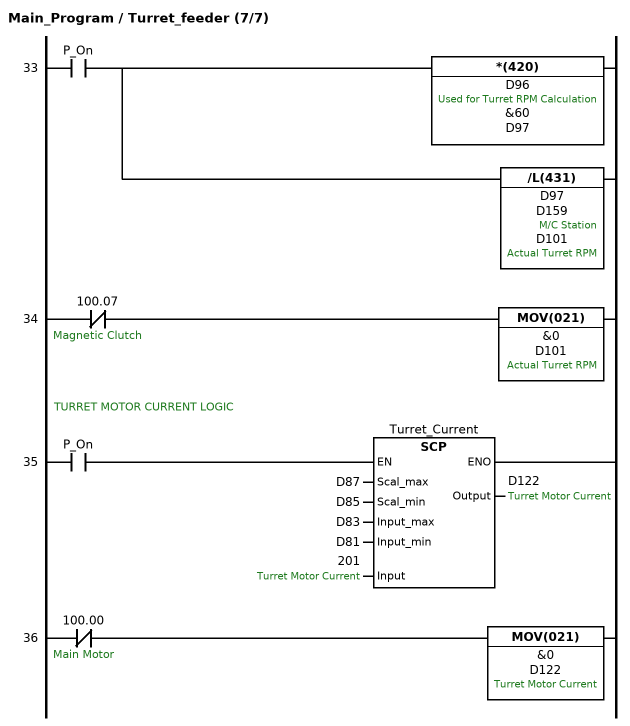
; [picture p24: Main_Program / Turret_feeder, rungs 33-36]
; rung 33
LD P_On
*(420) D96 &60 D97  ; Used for Turret RPM Calculation
/L(431) D97 D159 D101  ; M/C Station, Actual Turret RPM
; rung 34
LDNOT 100.07  ; Magnetic Clutch
MOV(021) &0 D101  ; Actual Turret RPM
; rung 35: TURRET MOTOR CURRENT LOGIC
LD P_On
CALL Turret_Current : SCP (Scal_max := D87, Scal_min := D85, Input_max := D83, Input_min := D81, Input := 201, Output => D122)  ; Turret Motor Current
; rung 36
LDNOT 100.00  ; Main Motor
MOV(021) &0 D122  ; Turret Motor Current

### Section Hyd_System
; Main Hyd. System Pressure

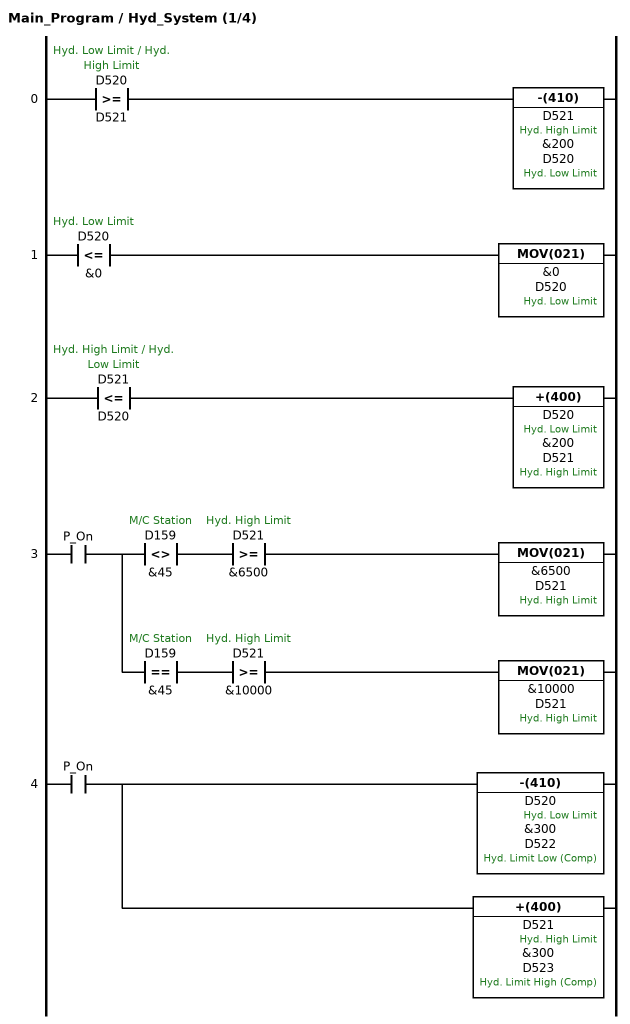
; rung 0
LD>=(325) D520 D521  ; Hyd. Low Limit, Hyd. High Limit
-(410) D521 &200 D520  ; Hyd. High Limit, Hyd. Low Limit
; rung 1
LD<=S(317) D520 &0  ; Hyd. Low Limit
MOV(021) &0 D520  ; Hyd. Low Limit
; rung 2
LD<=(315) D521 D520  ; Hyd. High Limit, Hyd. Low Limit
+(400) D520 &200 D521  ; Hyd. Low Limit, Hyd. High Limit
; rung 3
LD P_On
OUT TR0
AND<>(305) D159 &45  ; M/C Station
AND>=(325) D521 &6500  ; Hyd. High Limit
MOV(021) &6500 D521  ; Hyd. High Limit
LD TR0
AND=(300) D159 &45  ; M/C Station
AND>=(325) D521 &10000  ; Hyd. High Limit
MOV(021) &10000 D521  ; Hyd. High Limit
; rung 4
LD P_On
-(410) D520 &300 D522  ; Hyd. Low Limit, Hyd. Limit Low (Comp)
+(400) D521 &300 D523  ; Hyd. High Limit, Hyd. Limit High (Comp)

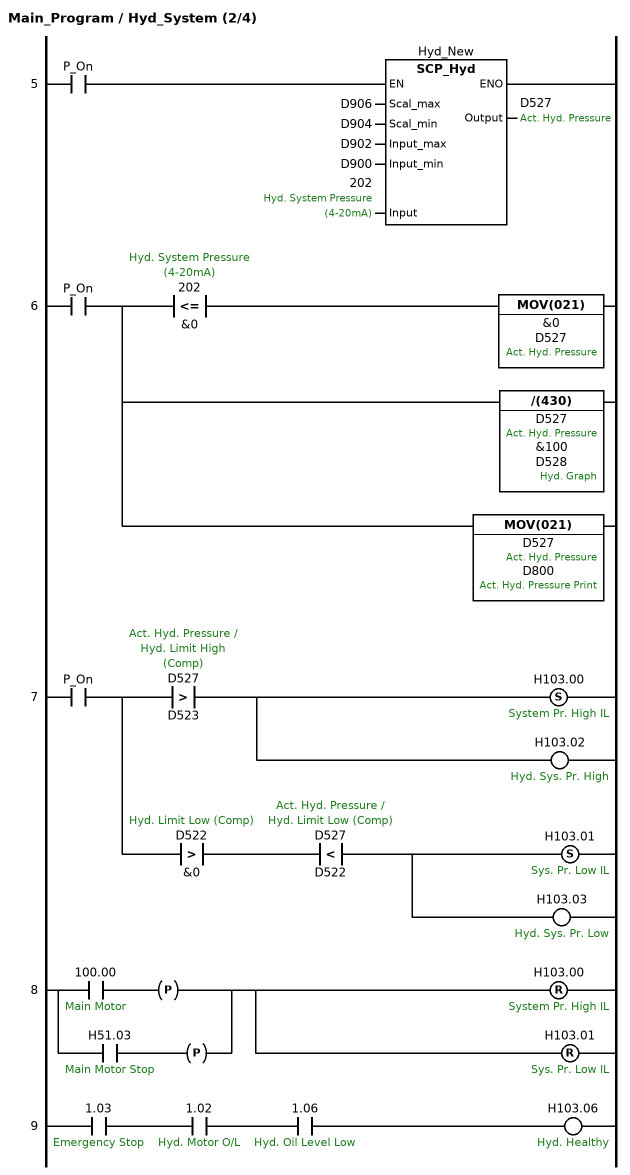
; rung 5
LD P_On
CALL Hyd_New : SCP_Hyd (Scal_max := D906, Scal_min := D904, Input_max := D902, Input_min := D900, Input := 202, Output => D527)  ; Hyd. System Pressure (4-20mA), Act. Hyd. Pressure
; rung 6
LD P_On
OUT TR0
AND<=S(317) 202 &0  ; Hyd. System Pressure (4-20mA)
MOV(021) &0 D527  ; Act. Hyd. Pressure
LD TR0
/(430) D527 &100 D528  ; Act. Hyd. Pressure, Hyd. Graph
MOV(021) D527 D800  ; Act. Hyd. Pressure, Act. Hyd. Pressure Print
; rung 7
LD P_On
OUT TR0
AND>(320) D527 D523  ; Act. Hyd. Pressure, Hyd. Limit High (Comp)
SET H103.00  ; System Pr. High IL
OUT H103.02  ; Hyd. Sys. Pr. High
LD TR0
AND>S(322) D522 &0  ; Hyd. Limit Low (Comp)
AND<(310) D527 D522  ; Act. Hyd. Pressure, Hyd. Limit Low (Comp)
SET H103.01  ; Sys. Pr. Low IL
OUT H103.03  ; Hyd. Sys. Pr. Low
; rung 8
LD 100.00  ; Main Motor
UP(521)
LD H51.03  ; Main Motor Stop
UP(521)
ORLD
RSET H103.00  ; System Pr. High IL
RSET H103.01  ; Sys. Pr. Low IL
; rung 9
LD 1.03  ; Emergency Stop
AND 1.02  ; Hyd. Motor O/L
AND 1.06  ; Hyd. Oil Level Low
OUT H103.06  ; Hyd. Healthy

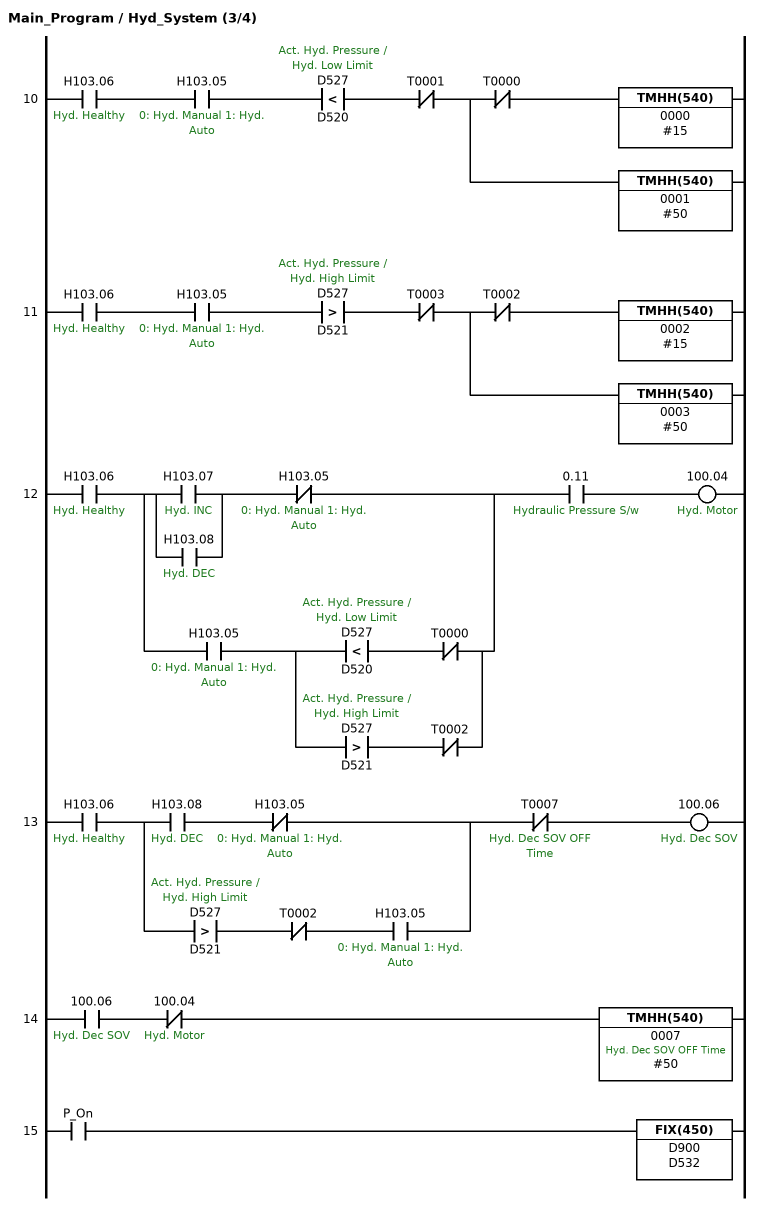
; rung 10
LD H103.06  ; Hyd. Healthy
AND H103.05  ; 0: Hyd. Manual 1: Hyd. Auto
AND<(310) D527 D520  ; Act. Hyd. Pressure, Hyd. Low Limit
ANDNOT T0001
OUT TR0
ANDNOT T0000
TMHH(540) 0000 #15
LD TR0
TMHH(540) 0001 #50
; rung 11
LD H103.06  ; Hyd. Healthy
AND H103.05  ; 0: Hyd. Manual 1: Hyd. Auto
AND>(320) D527 D521  ; Act. Hyd. Pressure, Hyd. High Limit
ANDNOT T0003
OUT TR0
ANDNOT T0002
TMHH(540) 0002 #15
LD TR0
TMHH(540) 0003 #50
; rung 12
LD H103.06  ; Hyd. Healthy
LD H103.07  ; Hyd. INC
OR H103.08  ; Hyd. DEC
ANDNOT H103.05  ; 0: Hyd. Manual 1: Hyd. Auto
LD H103.05  ; 0: Hyd. Manual 1: Hyd. Auto
LD<(310) D527 D520  ; Act. Hyd. Pressure, Hyd. Low Limit
ANDNOT T0000
LD>(320) D527 D521  ; Act. Hyd. Pressure, Hyd. High Limit
ANDNOT T0002
ORLD
ANDLD
ORLD
ANDLD
AND 0.11  ; Hydraulic Pressure S/w
OUT 100.04  ; Hyd. Motor
; rung 13
LD H103.06  ; Hyd. Healthy
LD H103.08  ; Hyd. DEC
ANDNOT H103.05  ; 0: Hyd. Manual 1: Hyd. Auto
LD>(320) D527 D521  ; Act. Hyd. Pressure, Hyd. High Limit
ANDNOT T0002
AND H103.05  ; 0: Hyd. Manual 1: Hyd. Auto
ORLD
ANDLD
ANDNOT T0007  ; Hyd. Dec SOV OFF Time
OUT 100.06  ; Hyd. Dec SOV
; rung 14
LD 100.06  ; Hyd. Dec SOV
ANDNOT 100.04  ; Hyd. Motor
TMHH(540) 0007 #50  ; Hyd. Dec SOV OFF Time
; rung 15
LD P_On
FIX(450) D900 D532

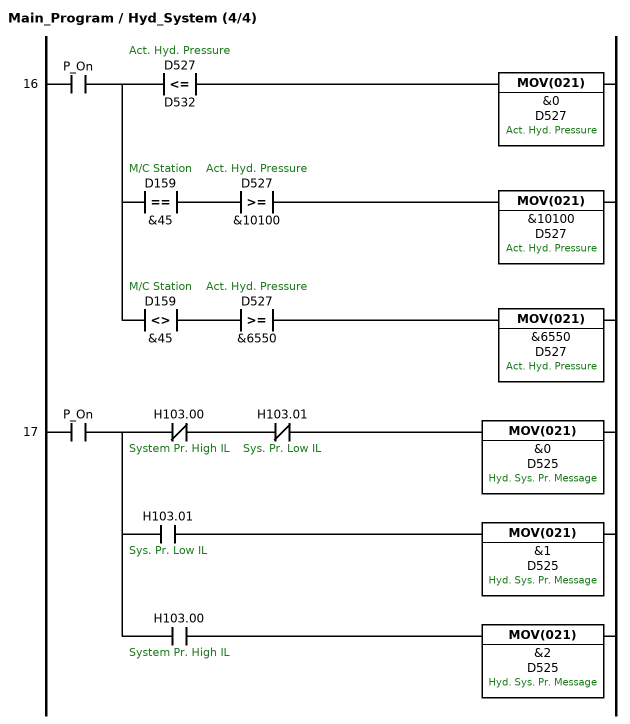
; rung 16
LD P_On
OUT TR0
AND<=(315) D527 D532  ; Act. Hyd. Pressure
MOV(021) &0 D527  ; Act. Hyd. Pressure
LD TR0
AND=(300) D159 &45  ; M/C Station
AND>=(325) D527 &10100  ; Act. Hyd. Pressure
MOV(021) &10100 D527  ; Act. Hyd. Pressure
LD TR0
AND<>(305) D159 &45  ; M/C Station
AND>=(325) D527 &6550  ; Act. Hyd. Pressure
MOV(021) &6550 D527  ; Act. Hyd. Pressure
; rung 17
LD P_On
OUT TR0
ANDNOT H103.00  ; System Pr. High IL
ANDNOT H103.01  ; Sys. Pr. Low IL
MOV(021) &0 D525  ; Hyd. Sys. Pr. Message
LD TR0
AND H103.01  ; Sys. Pr. Low IL
MOV(021) &1 D525  ; Hyd. Sys. Pr. Message
LD TR0
AND H103.00  ; System Pr. High IL
MOV(021) &2 D525  ; Hyd. Sys. Pr. Message

### Section Lubrication
; Lubrication Control & Hour Meter

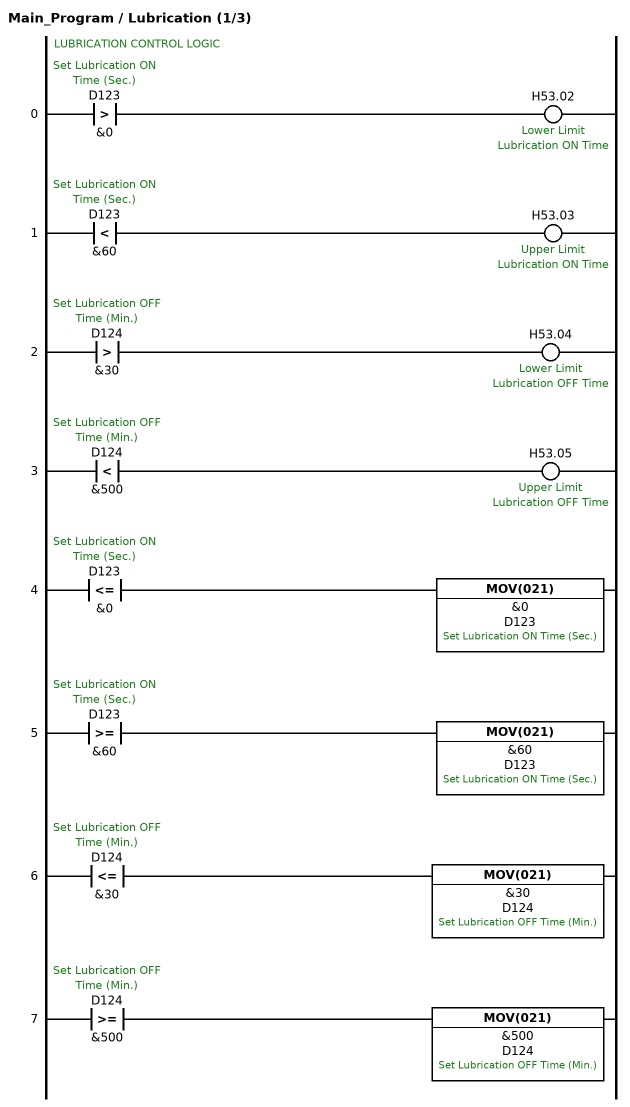
; rung 0: LUBRICATION CONTROL LOGIC
LD>(320) D123 &0  ; Set Lubrication ON Time (Sec.)
OUT H53.02  ; Lower Limit Lubrication ON Time
; rung 1
LD<(310) D123 &60  ; Set Lubrication ON Time (Sec.)
OUT H53.03  ; Upper Limit Lubrication ON Time
; rung 2
LD>(320) D124 &30  ; Set Lubrication OFF Time (Min.)
OUT H53.04  ; Lower Limit Lubrication OFF Time
; rung 3
LD<(310) D124 &500  ; Set Lubrication OFF Time (Min.)
OUT H53.05  ; Upper Limit Lubrication OFF Time
; rung 4
LD<=(315) D123 &0  ; Set Lubrication ON Time (Sec.)
MOV(021) &0 D123  ; Set Lubrication ON Time (Sec.)
; rung 5
LD>=(325) D123 &60  ; Set Lubrication ON Time (Sec.)
MOV(021) &60 D123  ; Set Lubrication ON Time (Sec.)
; rung 6
LD<=(315) D124 &30  ; Set Lubrication OFF Time (Min.)
MOV(021) &30 D124  ; Set Lubrication OFF Time (Min.)
; rung 7
LD>=(325) D124 &500  ; Set Lubrication OFF Time (Min.)
MOV(021) &500 D124  ; Set Lubrication OFF Time (Min.)

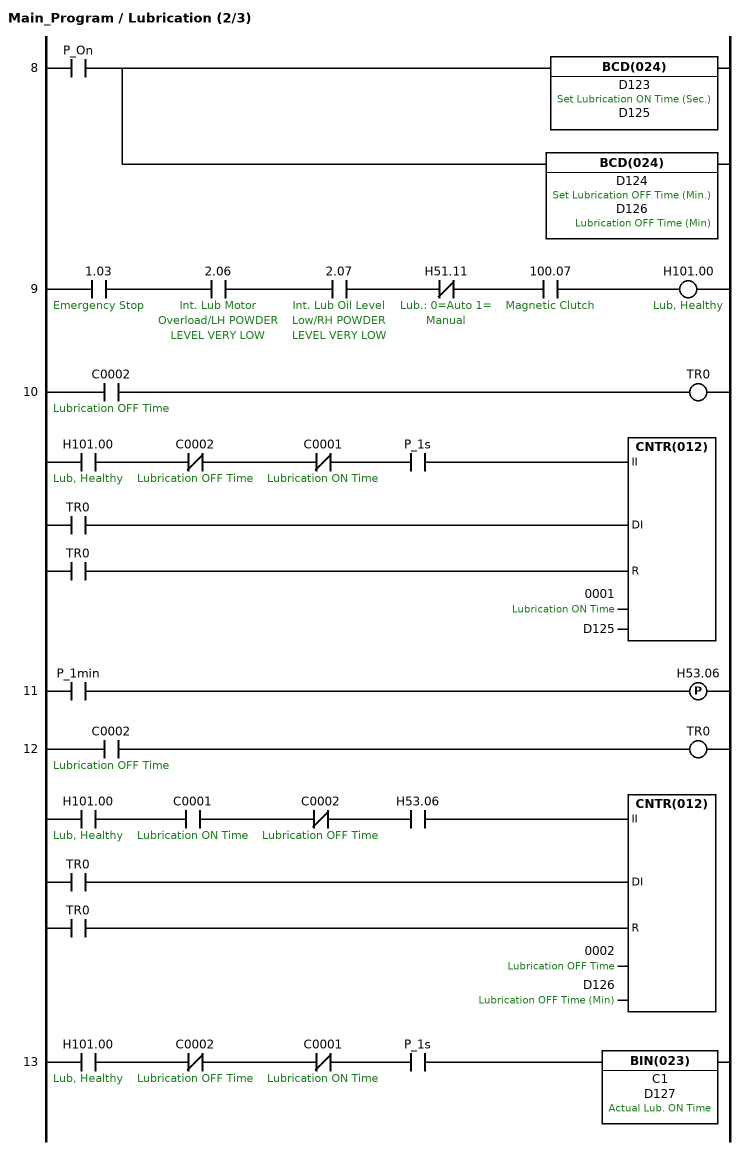
; rung 8
LD P_On
BCD(024) D123 D125  ; Set Lubrication ON Time (Sec.)
BCD(024) D124 D126  ; Set Lubrication OFF Time (Min.), Lubrication OFF Time (Min)
; rung 9
LD 1.03  ; Emergency Stop
AND 2.06  ; Int. Lub Motor Overload/LH POWDER LEVEL VERY LOW
AND 2.07  ; Int. Lub Oil Level Low/RH POWDER LEVEL VERY LOW
ANDNOT H51.11  ; Lub.: 0=Auto 1= Manual
AND 100.07  ; Magnetic Clutch
OUT H101.00  ; Lub, Healthy
; rung 10
LD H101.00  ; Lub, Healthy
ANDNOT C0002  ; Lubrication OFF Time
ANDNOT C0001  ; Lubrication ON Time
AND P_1s
LD C0002  ; Lubrication OFF Time
OUT TR0
LD TR0
CNTR(012) 0001 D125  ; Lubrication ON Time
; rung 11
LD P_1min
DIFU(013) H53.06
; rung 12
LD H101.00  ; Lub, Healthy
AND C0001  ; Lubrication ON Time
ANDNOT C0002  ; Lubrication OFF Time
AND H53.06
LD C0002  ; Lubrication OFF Time
OUT TR0
LD TR0
CNTR(012) 0002 D126  ; Lubrication OFF Time (Min), Lubrication OFF Time
; rung 13
LD H101.00  ; Lub, Healthy
ANDNOT C0002  ; Lubrication OFF Time
ANDNOT C0001  ; Lubrication ON Time
AND P_1s
BIN(023) C1 D127  ; Actual Lub. ON Time

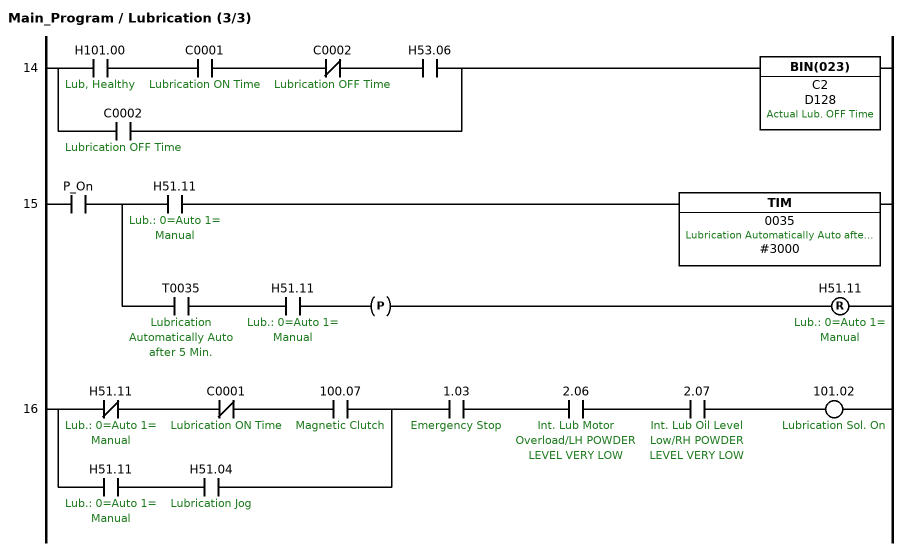
; rung 14
LD H101.00  ; Lub, Healthy
AND C0001  ; Lubrication ON Time
ANDNOT C0002  ; Lubrication OFF Time
AND H53.06
OR C0002  ; Lubrication OFF Time
BIN(023) C2 D128  ; Actual Lub. OFF Time
; rung 15
LD P_On
OUT TR0
AND H51.11  ; Lub.: 0=Auto 1= Manual
TIM 0035 #3000  ; Lubrication Automatically Auto after 5 Min.
LD TR0
AND T0035  ; Lubrication Automatically Auto after 5 Min.
AND H51.11  ; Lub.: 0=Auto 1= Manual
UP(521)
RSET H51.11  ; Lub.: 0=Auto 1= Manual
; rung 16
LDNOT H51.11  ; Lub.: 0=Auto 1= Manual
ANDNOT C0001  ; Lubrication ON Time
AND 100.07  ; Magnetic Clutch
LD H51.11  ; Lub.: 0=Auto 1= Manual
AND H51.04  ; Lubrication Jog
ORLD
AND 1.03  ; Emergency Stop
AND 2.06  ; Int. Lub Motor Overload/LH POWDER LEVEL VERY LOW
AND 2.07  ; Int. Lub Oil Level Low/RH POWDER LEVEL VERY LOW
OUT 101.02  ; Lubrication Sol. On

### Section LPSL
; Lower Punch Spray Control

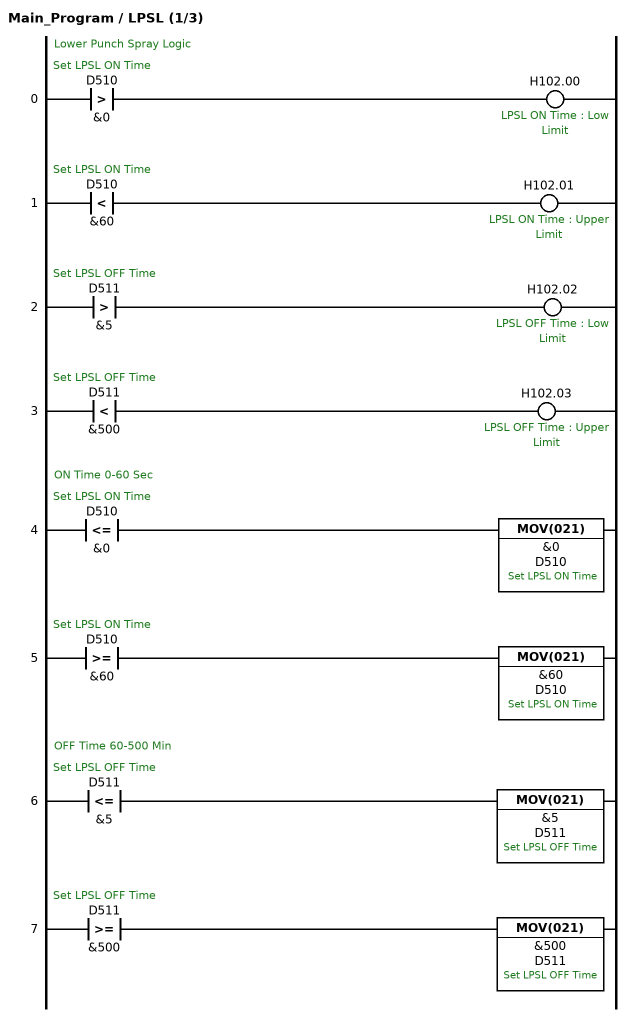
; rung 0: Lower Punch Spray Logic
LD>(320) D510 &0  ; Set LPSL ON Time
OUT H102.00  ; LPSL ON Time : Low Limit
; rung 1
LD<(310) D510 &60  ; Set LPSL ON Time
OUT H102.01  ; LPSL ON Time : Upper Limit
; rung 2
LD>(320) D511 &5  ; Set LPSL OFF Time
OUT H102.02  ; LPSL OFF Time : Low Limit
; rung 3
LD<(310) D511 &500  ; Set LPSL OFF Time
OUT H102.03  ; LPSL OFF Time : Upper Limit
; rung 4: ON Time 0-60 Sec
LD<=(315) D510 &0  ; Set LPSL ON Time
MOV(021) &0 D510  ; Set LPSL ON Time
; rung 5
LD>=(325) D510 &60  ; Set LPSL ON Time
MOV(021) &60 D510  ; Set LPSL ON Time
; rung 6: OFF Time 60-500 Min
LD<=(315) D511 &5  ; Set LPSL OFF Time
MOV(021) &5 D511  ; Set LPSL OFF Time
; rung 7
LD>=(325) D511 &500  ; Set LPSL OFF Time
MOV(021) &500 D511  ; Set LPSL OFF Time

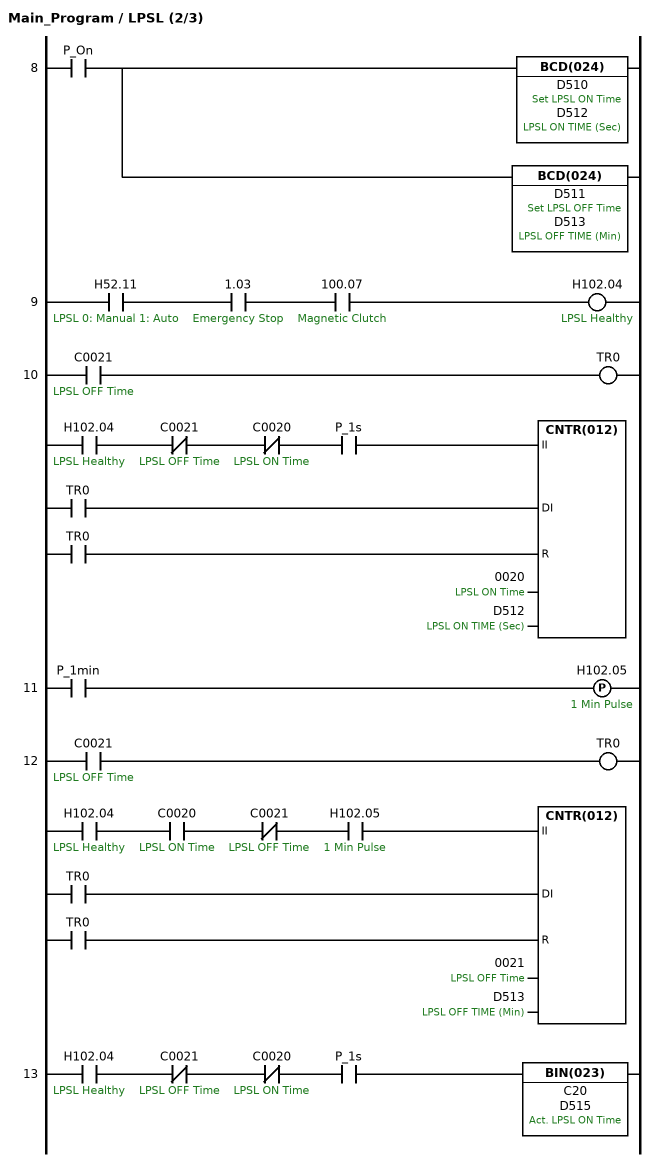
; rung 8
LD P_On
BCD(024) D510 D512  ; Set LPSL ON Time, LPSL ON TIME (Sec)
BCD(024) D511 D513  ; Set LPSL OFF Time, LPSL OFF TIME (Min)
; rung 9
LD H52.11  ; LPSL 0: Manual 1: Auto
AND 1.03  ; Emergency Stop
AND 100.07  ; Magnetic Clutch
OUT H102.04  ; LPSL Healthy
; rung 10
LD H102.04  ; LPSL Healthy
ANDNOT C0021  ; LPSL OFF Time
ANDNOT C0020  ; LPSL ON Time
AND P_1s
LD C0021  ; LPSL OFF Time
OUT TR0
LD TR0
CNTR(012) 0020 D512  ; LPSL ON TIME (Sec), LPSL ON Time
; rung 11
LD P_1min
DIFU(013) H102.05  ; 1 Min Pulse
; rung 12
LD H102.04  ; LPSL Healthy
AND C0020  ; LPSL ON Time
ANDNOT C0021  ; LPSL OFF Time
AND H102.05  ; 1 Min Pulse
LD C0021  ; LPSL OFF Time
OUT TR0
LD TR0
CNTR(012) 0021 D513  ; LPSL OFF TIME (Min), LPSL OFF Time
; rung 13
LD H102.04  ; LPSL Healthy
ANDNOT C0021  ; LPSL OFF Time
ANDNOT C0020  ; LPSL ON Time
AND P_1s
BIN(023) C20 D515  ; Act. LPSL ON Time

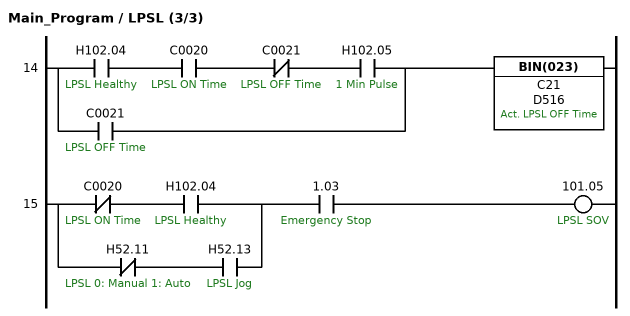
; rung 14
LD H102.04  ; LPSL Healthy
AND C0020  ; LPSL ON Time
ANDNOT C0021  ; LPSL OFF Time
AND H102.05  ; 1 Min Pulse
OR C0021  ; LPSL OFF Time
BIN(023) C21 D516  ; Act. LPSL OFF Time
; rung 15
LDNOT C0020  ; LPSL ON Time
AND H102.04  ; LPSL Healthy
LDNOT H52.11  ; LPSL 0: Manual 1: Auto
AND H52.13  ; LPSL Jog
ORLD
AND 1.03  ; Emergency Stop
OUT 101.05  ; LPSL SOV

### Section Agitator

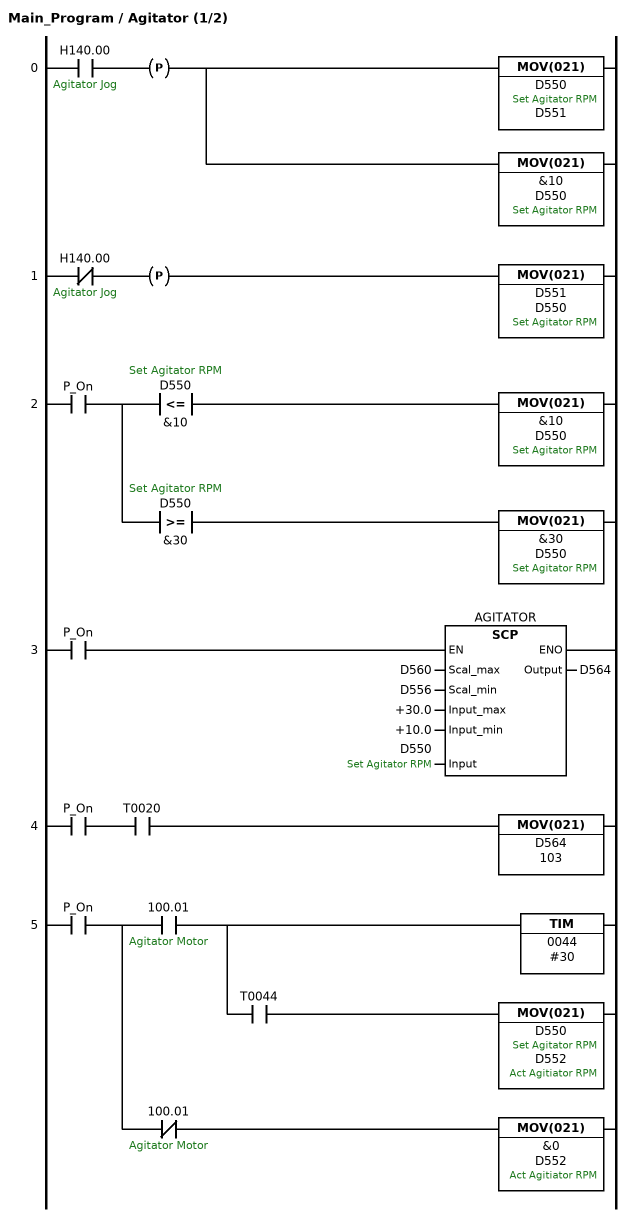
; rung 0
LD H140.00  ; Agitator Jog
UP(521)
MOV(021) D550 D551  ; Set Agitator RPM
MOV(021) &10 D550  ; Set Agitator RPM
; rung 1
LDNOT H140.00  ; Agitator Jog
UP(521)
MOV(021) D551 D550  ; Set Agitator RPM
; rung 2
LD P_On
OUT TR0
AND<=(315) D550 &10  ; Set Agitator RPM
MOV(021) &10 D550  ; Set Agitator RPM
LD TR0
AND>=(325) D550 &30  ; Set Agitator RPM
MOV(021) &30 D550  ; Set Agitator RPM
; rung 3
LD P_On
CALL AGITATOR : SCP (Scal_max := D560, Scal_min := D556, Input_max := +30.0, Input_min := +10.0, Input := D550, Output => D564)  ; Set Agitator RPM
; rung 4
LD P_On
AND T0020
MOV(021) D564 103
; rung 5
LD P_On
OUT TR0
AND 100.01  ; Agitator Motor
TIM 0044 #30
AND T0044
MOV(021) D550 D552  ; Set Agitator RPM, Act Agitiator RPM
LD TR0
ANDNOT 100.01  ; Agitator Motor
MOV(021) &0 D552  ; Act Agitiator RPM

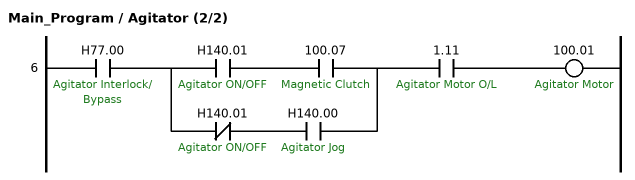
; rung 6
LD H77.00  ; Agitator Interlock/Bypass
LD H140.01  ; Agitator ON/OFF
AND 100.07  ; Magnetic Clutch
LDNOT H140.01  ; Agitator ON/OFF
AND H140.00  ; Agitator Jog
ORLD
ANDLD
AND 1.11  ; Agitator Motor O/L
OUT 100.01  ; Agitator Motor

### Section Recipe

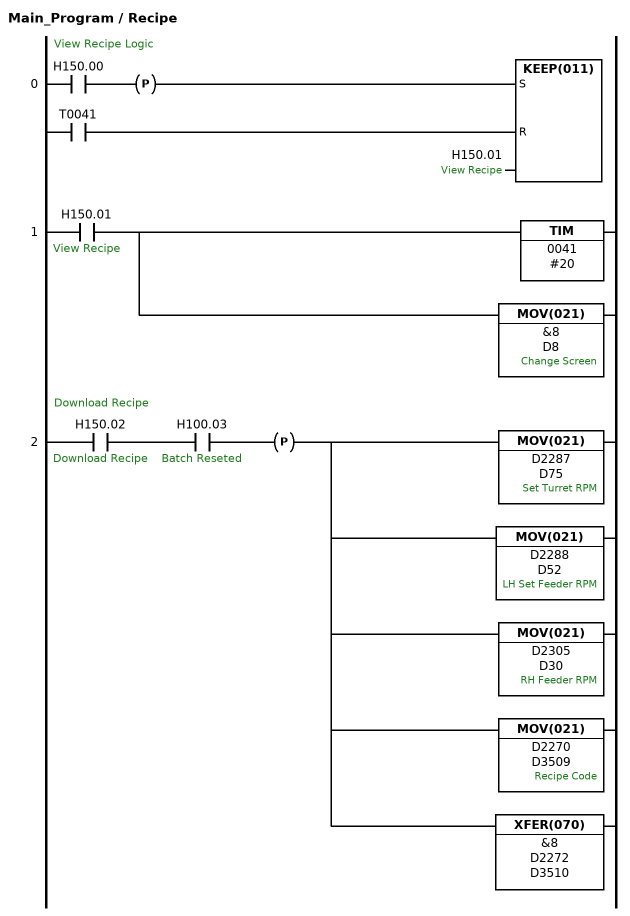
; rung 0: View Recipe Logic
LD H150.00
UP(521)
LD T0041
KEEP(011) H150.01  ; View Recipe
; rung 1
LD H150.01  ; View Recipe
TIM 0041 #20
MOV(021) &8 D8  ; Change Screen
; rung 2: Download Recipe
LD H150.02  ; Download Recipe
AND H100.03  ; Batch Reseted
UP(521)
MOV(021) D2287 D75  ; Set Turret RPM
MOV(021) D2288 D52  ; LH Set Feeder RPM
MOV(021) D2305 D30  ; RH Feeder RPM
MOV(021) D2270 D3509  ; Recipe Code
XFER(070) &8 D2272 D3510

### Section Interlock

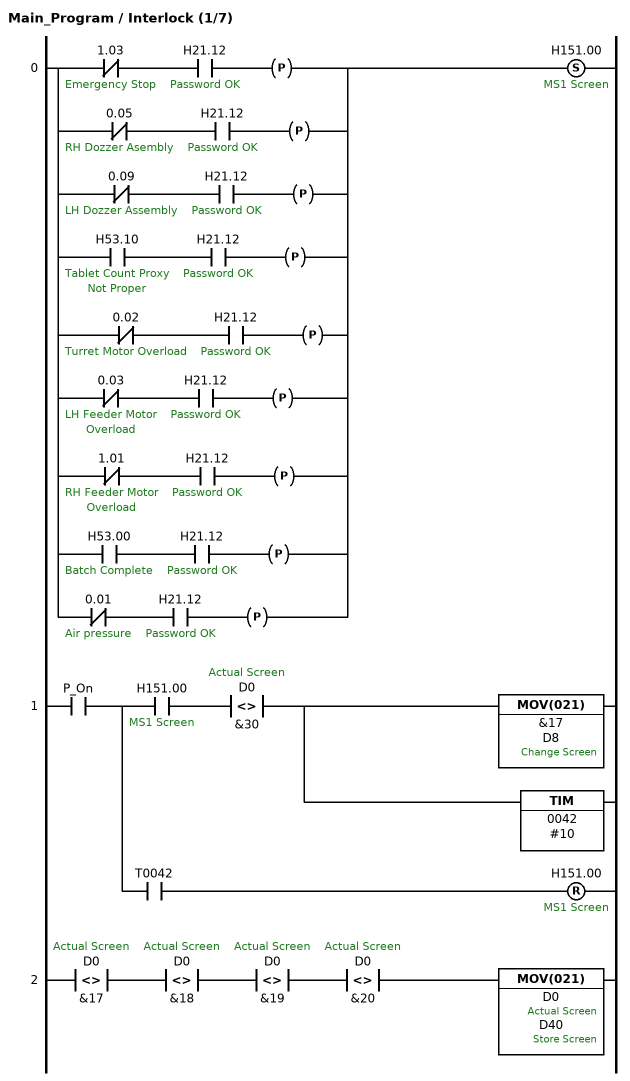
; rung 0
LDNOT 1.03  ; Emergency Stop
AND H21.12  ; Password OK
UP(521)
LDNOT 0.05  ; RH Dozzer Asembly
AND H21.12  ; Password OK
UP(521)
ORLD
LDNOT 0.09  ; LH Dozzer Assembly
AND H21.12  ; Password OK
UP(521)
ORLD
LD H53.10  ; Tablet Count Proxy Not Proper
AND H21.12  ; Password OK
UP(521)
ORLD
LDNOT 0.02  ; Turret Motor Overload
AND H21.12  ; Password OK
UP(521)
ORLD
LDNOT 0.03  ; LH Feeder Motor Overload
AND H21.12  ; Password OK
UP(521)
ORLD
LDNOT 1.01  ; RH Feeder Motor Overload
AND H21.12  ; Password OK
UP(521)
ORLD
LD H53.00  ; Batch Complete
AND H21.12  ; Password OK
UP(521)
ORLD
LDNOT 0.01  ; Air pressure
AND H21.12  ; Password OK
UP(521)
ORLD
SET H151.00  ; MS1 Screen
; rung 1
LD P_On
OUT TR0
AND H151.00  ; MS1 Screen
AND<>(305) D0 &30  ; Actual Screen
MOV(021) &17 D8  ; Change Screen
TIM 0042 #10
LD TR0
AND T0042
RSET H151.00  ; MS1 Screen
; rung 2
LD<>(305) D0 &17  ; Actual Screen
AND<>(305) D0 &18  ; Actual Screen
AND<>(305) D0 &19  ; Actual Screen
AND<>(305) D0 &20  ; Actual Screen
MOV(021) D0 D40  ; Actual Screen, Store Screen

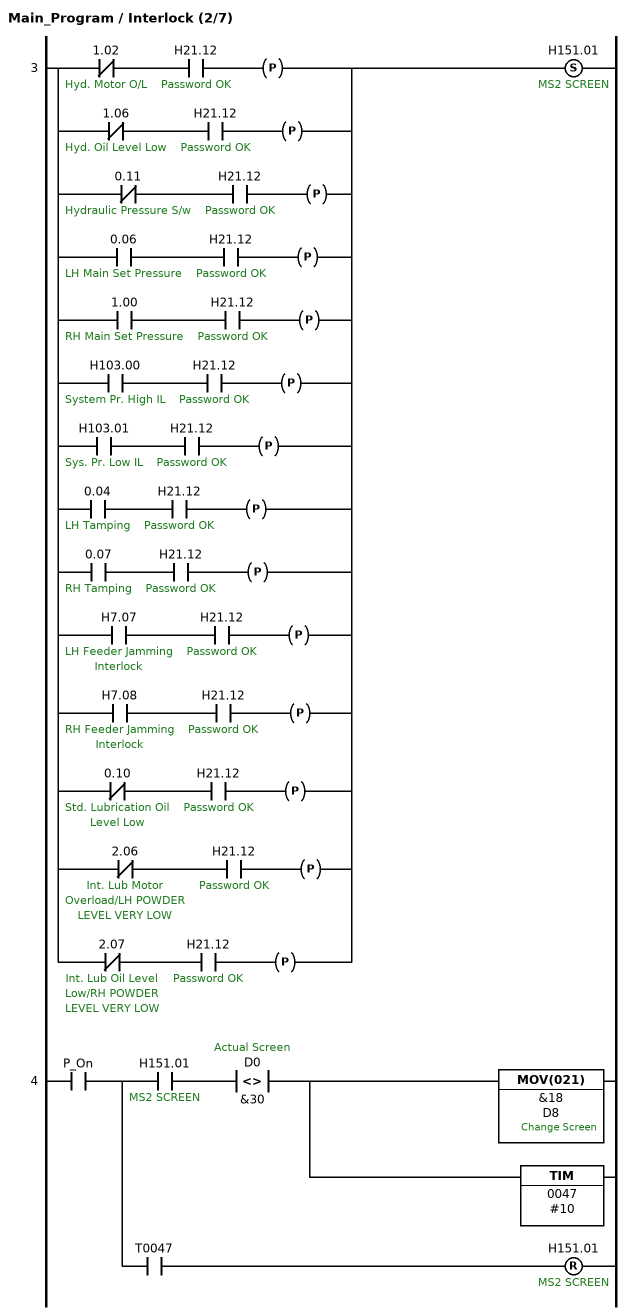
; rung 3
LDNOT 1.02  ; Hyd. Motor O/L
AND H21.12  ; Password OK
UP(521)
LDNOT 1.06  ; Hyd. Oil Level Low
AND H21.12  ; Password OK
UP(521)
ORLD
LDNOT 0.11  ; Hydraulic Pressure S/w
AND H21.12  ; Password OK
UP(521)
ORLD
LD 0.06  ; LH Main Set Pressure
AND H21.12  ; Password OK
UP(521)
ORLD
LD 1.00  ; RH Main Set Pressure
AND H21.12  ; Password OK
UP(521)
ORLD
LD H103.00  ; System Pr. High IL
AND H21.12  ; Password OK
UP(521)
ORLD
LD H103.01  ; Sys. Pr. Low IL
AND H21.12  ; Password OK
UP(521)
ORLD
LD 0.04  ; LH Tamping
AND H21.12  ; Password OK
UP(521)
ORLD
LD 0.07  ; RH Tamping
AND H21.12  ; Password OK
UP(521)
ORLD
LD H7.07  ; LH Feeder Jamming Interlock
AND H21.12  ; Password OK
UP(521)
ORLD
LD H7.08  ; RH Feeder Jamming Interlock
AND H21.12  ; Password OK
UP(521)
ORLD
LDNOT 0.10  ; Std. Lubrication Oil Level Low
AND H21.12  ; Password OK
UP(521)
ORLD
LDNOT 2.06  ; Int. Lub Motor Overload/LH POWDER LEVEL VERY LOW
AND H21.12  ; Password OK
UP(521)
ORLD
LDNOT 2.07  ; Int. Lub Oil Level Low/RH POWDER LEVEL VERY LOW
AND H21.12  ; Password OK
UP(521)
ORLD
SET H151.01  ; MS2 SCREEN
; rung 4
LD P_On
OUT TR0
AND H151.01  ; MS2 SCREEN
AND<>(305) D0 &30  ; Actual Screen
MOV(021) &18 D8  ; Change Screen
TIM 0047 #10
LD TR0
AND T0047
RSET H151.01  ; MS2 SCREEN

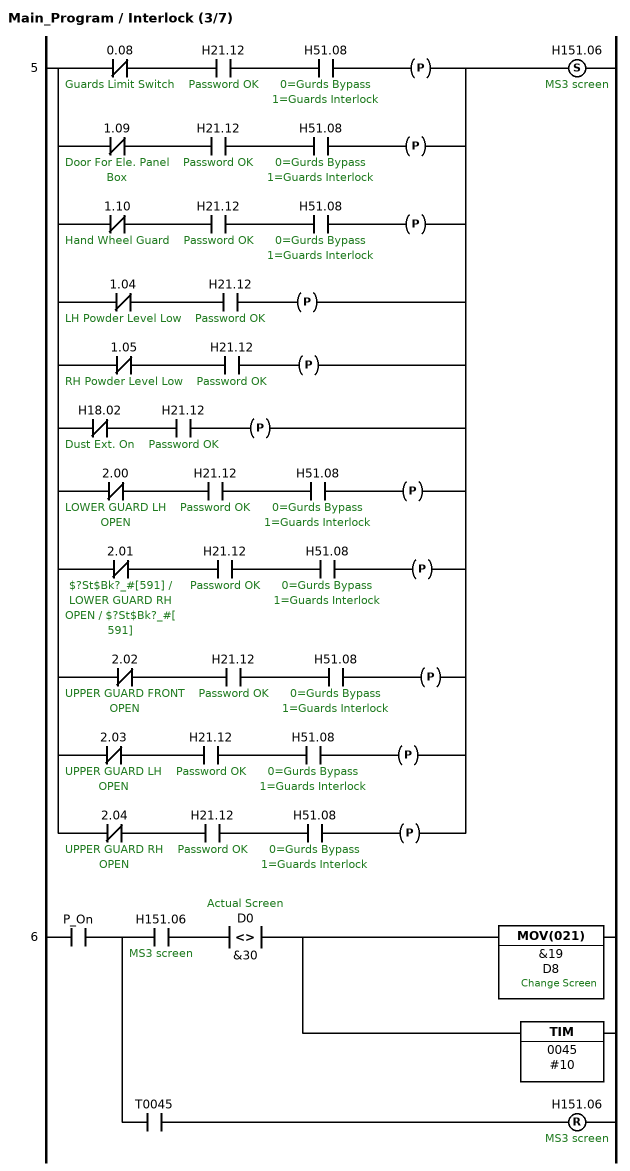
; rung 5
LDNOT 0.08  ; Guards Limit Switch
AND H21.12  ; Password OK
AND H51.08  ; 0=Gurds Bypass 1=Guards Interlock
UP(521)
LDNOT 1.09  ; Door For Ele. Panel Box
AND H21.12  ; Password OK
AND H51.08  ; 0=Gurds Bypass 1=Guards Interlock
UP(521)
ORLD
LDNOT 1.10  ; Hand Wheel Guard
AND H21.12  ; Password OK
AND H51.08  ; 0=Gurds Bypass 1=Guards Interlock
UP(521)
ORLD
LDNOT 1.04  ; LH Powder Level Low
AND H21.12  ; Password OK
UP(521)
ORLD
LDNOT 1.05  ; RH Powder Level Low
AND H21.12  ; Password OK
UP(521)
ORLD
LDNOT H18.02  ; Dust Ext. On
AND H21.12  ; Password OK
UP(521)
ORLD
LDNOT 2.00  ; LOWER GUARD LH OPEN
AND H21.12  ; Password OK
AND H51.08  ; 0=Gurds Bypass 1=Guards Interlock
UP(521)
ORLD
LDNOT 2.01  ; $?St$Bk?_#[591] / LOWER GUARD RH OPEN / $?St$Bk?_#[591]
AND H21.12  ; Password OK
AND H51.08  ; 0=Gurds Bypass 1=Guards Interlock
UP(521)
ORLD
LDNOT 2.02  ; UPPER GUARD FRONT OPEN
AND H21.12  ; Password OK
AND H51.08  ; 0=Gurds Bypass 1=Guards Interlock
UP(521)
ORLD
LDNOT 2.03  ; UPPER GUARD LH OPEN
AND H21.12  ; Password OK
AND H51.08  ; 0=Gurds Bypass 1=Guards Interlock
UP(521)
ORLD
LDNOT 2.04  ; UPPER GUARD RH OPEN
AND H21.12  ; Password OK
AND H51.08  ; 0=Gurds Bypass 1=Guards Interlock
UP(521)
ORLD
SET H151.06  ; MS3 screen
; rung 6
LD P_On
OUT TR0
AND H151.06  ; MS3 screen
AND<>(305) D0 &30  ; Actual Screen
MOV(021) &19 D8  ; Change Screen
TIM 0045 #10
LD TR0
AND T0045
RSET H151.06  ; MS3 screen

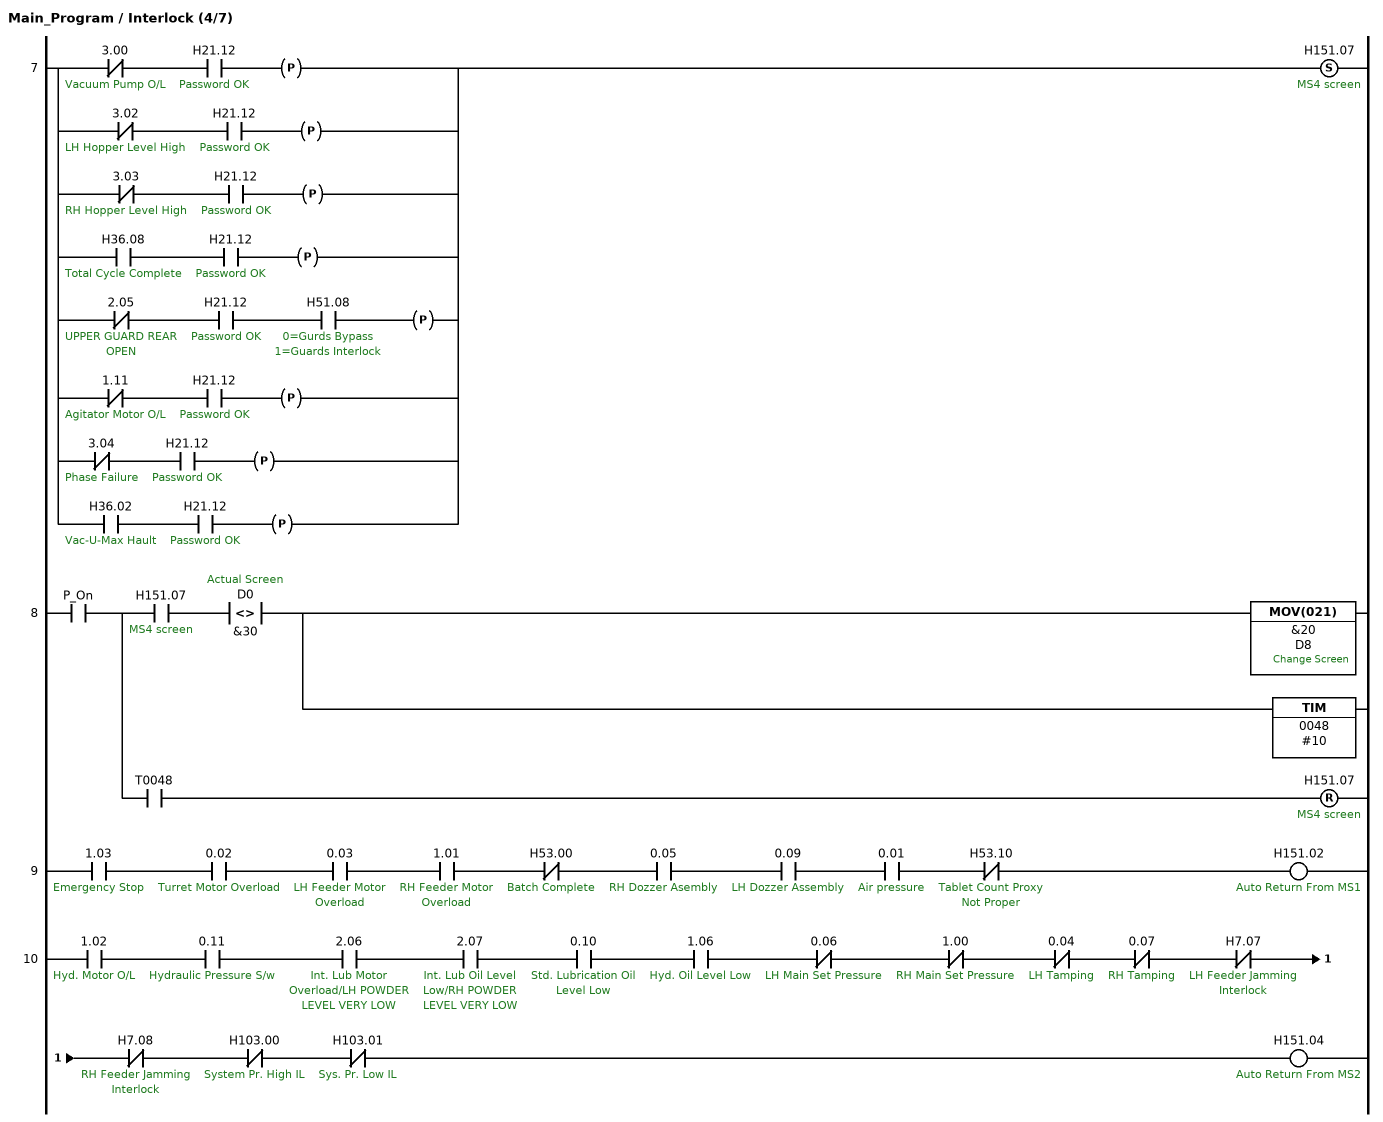
; rung 7
LDNOT 3.00  ; Vacuum Pump O/L
AND H21.12  ; Password OK
UP(521)
LDNOT 3.02  ; LH Hopper Level High
AND H21.12  ; Password OK
UP(521)
ORLD
LDNOT 3.03  ; RH Hopper Level High
AND H21.12  ; Password OK
UP(521)
ORLD
LD H36.08  ; Total Cycle Complete
AND H21.12  ; Password OK
UP(521)
ORLD
LDNOT 2.05  ; UPPER GUARD REAR OPEN
AND H21.12  ; Password OK
AND H51.08  ; 0=Gurds Bypass 1=Guards Interlock
UP(521)
ORLD
LDNOT 1.11  ; Agitator Motor O/L
AND H21.12  ; Password OK
UP(521)
ORLD
LDNOT 3.04  ; Phase Failure
AND H21.12  ; Password OK
UP(521)
ORLD
LD H36.02  ; Vac-U-Max Hault
AND H21.12  ; Password OK
UP(521)
ORLD
SET H151.07  ; MS4 screen
; rung 8
LD P_On
OUT TR0
AND H151.07  ; MS4 screen
AND<>(305) D0 &30  ; Actual Screen
MOV(021) &20 D8  ; Change Screen
TIM 0048 #10
LD TR0
AND T0048
RSET H151.07  ; MS4 screen
; rung 9
LD 1.03  ; Emergency Stop
AND 0.02  ; Turret Motor Overload
AND 0.03  ; LH Feeder Motor Overload
AND 1.01  ; RH Feeder Motor Overload
ANDNOT H53.00  ; Batch Complete
AND 0.05  ; RH Dozzer Asembly
AND 0.09  ; LH Dozzer Assembly
AND 0.01  ; Air pressure
ANDNOT H53.10  ; Tablet Count Proxy Not Proper
OUT H151.02  ; Auto Return From MS1
; rung 10
LD 1.02  ; Hyd. Motor O/L
AND 0.11  ; Hydraulic Pressure S/w
AND 2.06  ; Int. Lub Motor Overload/LH POWDER LEVEL VERY LOW
AND 2.07  ; Int. Lub Oil Level Low/RH POWDER LEVEL VERY LOW
AND 0.10  ; Std. Lubrication Oil Level Low
AND 1.06  ; Hyd. Oil Level Low
ANDNOT 0.06  ; LH Main Set Pressure
ANDNOT 1.00  ; RH Main Set Pressure
ANDNOT 0.04  ; LH Tamping
ANDNOT 0.07  ; RH Tamping
ANDNOT H7.07  ; LH Feeder Jamming Interlock
ANDNOT H7.08  ; RH Feeder Jamming Interlock
ANDNOT H103.00  ; System Pr. High IL
ANDNOT H103.01  ; Sys. Pr. Low IL
OUT H151.04  ; Auto Return From MS2

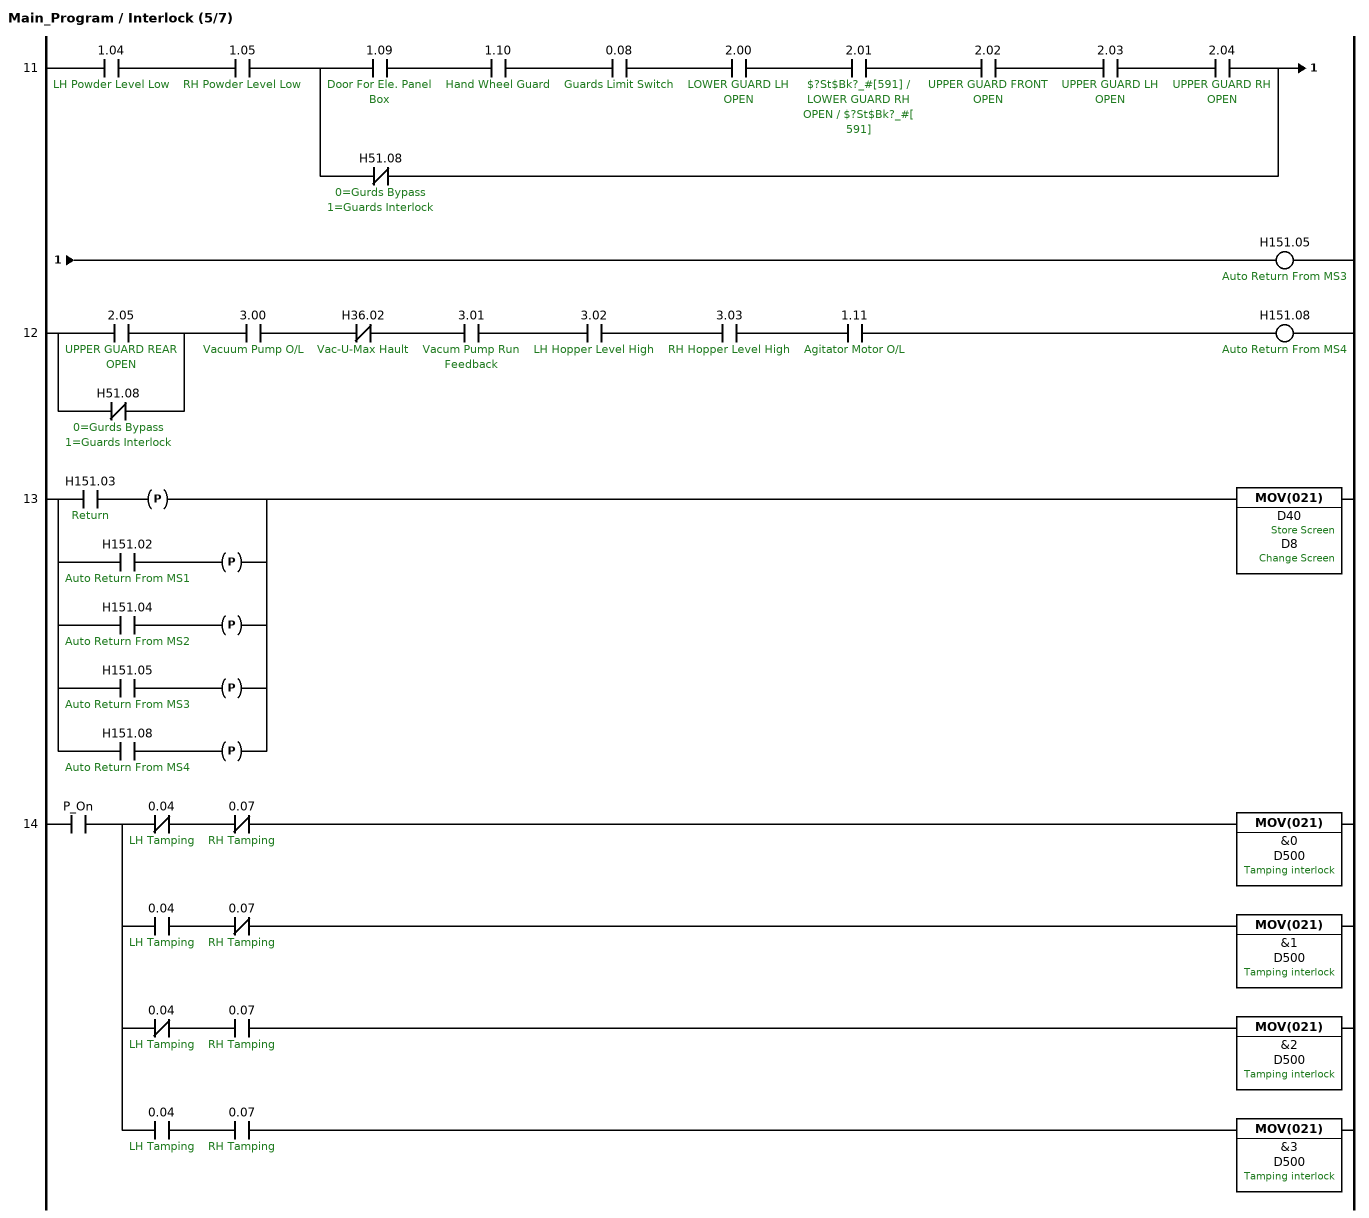
; rung 11
LD 1.04  ; LH Powder Level Low
AND 1.05  ; RH Powder Level Low
LD 1.09  ; Door For Ele. Panel Box
AND 1.10  ; Hand Wheel Guard
AND 0.08  ; Guards Limit Switch
AND 2.00  ; LOWER GUARD LH OPEN
AND 2.01  ; $?St$Bk?_#[591] / LOWER GUARD RH OPEN / $?St$Bk?_#[591]
AND 2.02  ; UPPER GUARD FRONT OPEN
AND 2.03  ; UPPER GUARD LH OPEN
AND 2.04  ; UPPER GUARD RH OPEN
ORNOT H51.08  ; 0=Gurds Bypass 1=Guards Interlock
ANDLD
OUT H151.05  ; Auto Return From MS3
; rung 12
LD 2.05  ; UPPER GUARD REAR OPEN
ORNOT H51.08  ; 0=Gurds Bypass 1=Guards Interlock
AND 3.00  ; Vacuum Pump O/L
ANDNOT H36.02  ; Vac-U-Max Hault
AND 3.01  ; Vacum Pump Run Feedback
AND 3.02  ; LH Hopper Level High
AND 3.03  ; RH Hopper Level High
AND 1.11  ; Agitator Motor O/L
OUT H151.08  ; Auto Return From MS4
; rung 13
LD H151.03  ; Return
UP(521)
LD H151.02  ; Auto Return From MS1
UP(521)
ORLD
LD H151.04  ; Auto Return From MS2
UP(521)
ORLD
LD H151.05  ; Auto Return From MS3
UP(521)
ORLD
LD H151.08  ; Auto Return From MS4
UP(521)
ORLD
MOV(021) D40 D8  ; Store Screen, Change Screen
; rung 14
LD P_On
OUT TR0
ANDNOT 0.04  ; LH Tamping
ANDNOT 0.07  ; RH Tamping
MOV(021) &0 D500  ; Tamping interlock
LD TR0
AND 0.04  ; LH Tamping
ANDNOT 0.07  ; RH Tamping
MOV(021) &1 D500  ; Tamping interlock
LD TR0
ANDNOT 0.04  ; LH Tamping
AND 0.07  ; RH Tamping
MOV(021) &2 D500  ; Tamping interlock
LD TR0
AND 0.04  ; LH Tamping
AND 0.07  ; RH Tamping
MOV(021) &3 D500  ; Tamping interlock

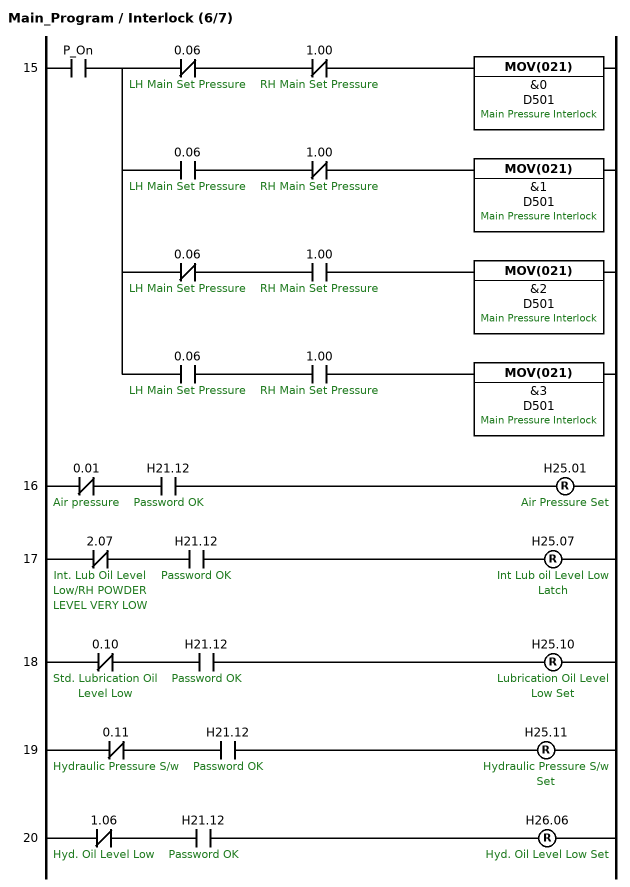
; rung 15
LD P_On
OUT TR0
ANDNOT 0.06  ; LH Main Set Pressure
ANDNOT 1.00  ; RH Main Set Pressure
MOV(021) &0 D501  ; Main Pressure Interlock
LD TR0
AND 0.06  ; LH Main Set Pressure
ANDNOT 1.00  ; RH Main Set Pressure
MOV(021) &1 D501  ; Main Pressure Interlock
LD TR0
ANDNOT 0.06  ; LH Main Set Pressure
AND 1.00  ; RH Main Set Pressure
MOV(021) &2 D501  ; Main Pressure Interlock
LD TR0
AND 0.06  ; LH Main Set Pressure
AND 1.00  ; RH Main Set Pressure
MOV(021) &3 D501  ; Main Pressure Interlock
; rung 16
LDNOT 0.01  ; Air pressure
AND H21.12  ; Password OK
RSET H25.01  ; Air Pressure Set
; rung 17
LDNOT 2.07  ; Int. Lub Oil Level Low/RH POWDER LEVEL VERY LOW
AND H21.12  ; Password OK
RSET H25.07  ; Int Lub oil Level Low Latch
; rung 18
LDNOT 0.10  ; Std. Lubrication Oil Level Low
AND H21.12  ; Password OK
RSET H25.10  ; Lubrication Oil Level Low Set
; rung 19
LDNOT 0.11  ; Hydraulic Pressure S/w
AND H21.12  ; Password OK
RSET H25.11  ; Hydraulic Pressure S/w Set
; rung 20
LDNOT 1.06  ; Hyd. Oil Level Low
AND H21.12  ; Password OK
RSET H26.06  ; Hyd. Oil Level Low Set

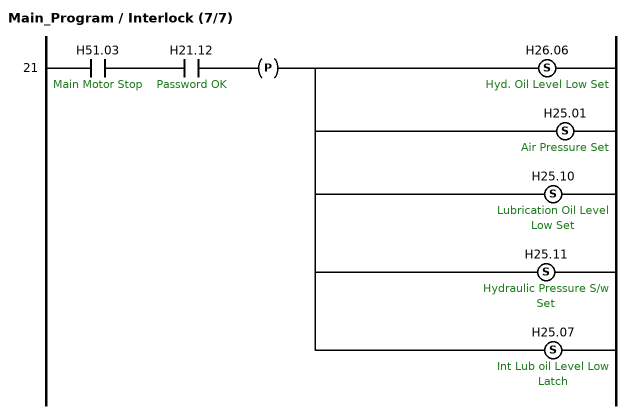
; rung 21
LD H51.03  ; Main Motor Stop
AND H21.12  ; Password OK
UP(521)
SET H26.06  ; Hyd. Oil Level Low Set
SET H25.01  ; Air Pressure Set
SET H25.10  ; Lubrication Oil Level Low Set
SET H25.11  ; Hydraulic Pressure S/w Set
SET H25.07  ; Int Lub oil Level Low Latch

### Section Feeder_Jamming

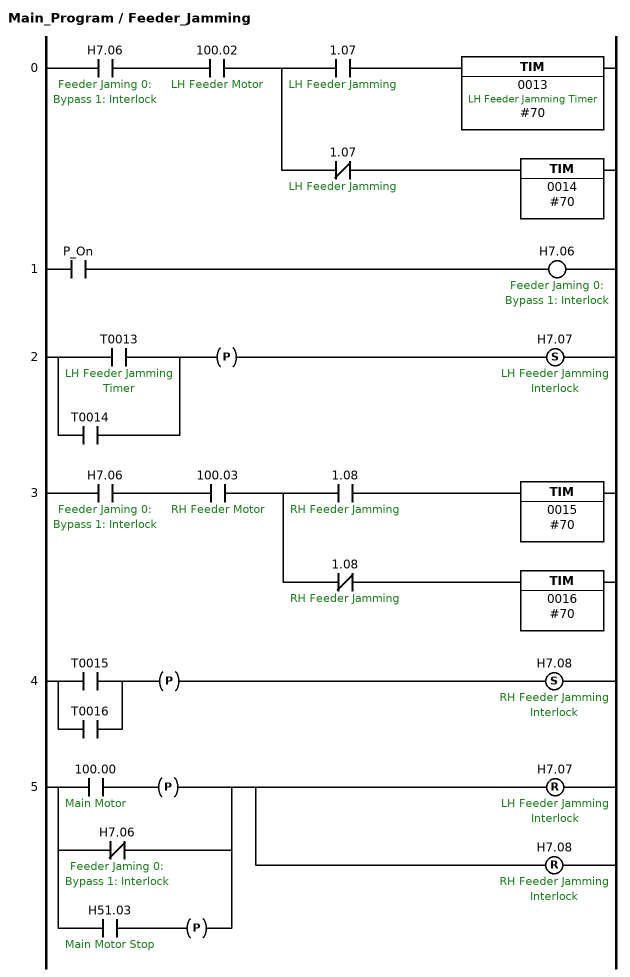
; rung 0
LD H7.06  ; Feeder Jaming 0: Bypass 1: Interlock
AND 100.02  ; LH Feeder Motor
OUT TR0
AND 1.07  ; LH Feeder Jamming
TIM 0013 #70  ; LH Feeder Jamming Timer
LD TR0
ANDNOT 1.07  ; LH Feeder Jamming
TIM 0014 #70
; rung 1
LD P_On
OUT H7.06  ; Feeder Jaming 0: Bypass 1: Interlock
; rung 2
LD T0013  ; LH Feeder Jamming Timer
OR T0014
UP(521)
SET H7.07  ; LH Feeder Jamming Interlock
; rung 3
LD H7.06  ; Feeder Jaming 0: Bypass 1: Interlock
AND 100.03  ; RH Feeder Motor
OUT TR0
AND 1.08  ; RH Feeder Jamming
TIM 0015 #70
LD TR0
ANDNOT 1.08  ; RH Feeder Jamming
TIM 0016 #70
; rung 4
LD T0015
OR T0016
UP(521)
SET H7.08  ; RH Feeder Jamming Interlock
; rung 5
LD 100.00  ; Main Motor
UP(521)
ORNOT H7.06  ; Feeder Jaming 0: Bypass 1: Interlock
LD H51.03  ; Main Motor Stop
UP(521)
ORLD
RSET H7.07  ; LH Feeder Jamming Interlock
RSET H7.08  ; RH Feeder Jamming Interlock

### Section Hour_meter

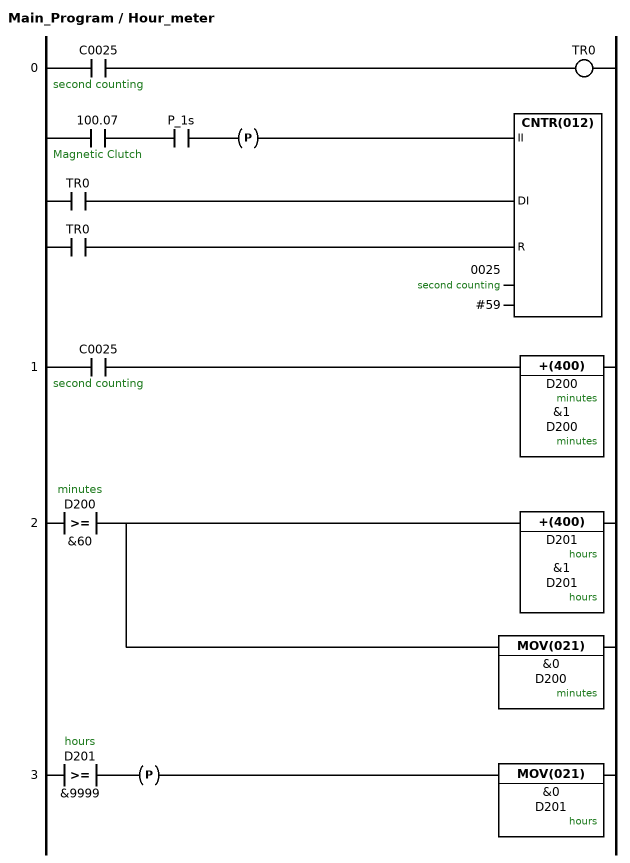
; rung 0
LD 100.07  ; Magnetic Clutch
AND P_1s
UP(521)
LD C0025  ; second counting
OUT TR0
LD TR0
CNTR(012) 0025 #59  ; second counting
; rung 1
LD C0025  ; second counting
+(400) D200 &1 D200  ; minutes
; rung 2
LD>=(325) D200 &60  ; minutes
+(400) D201 &1 D201  ; hours
MOV(021) &0 D200  ; minutes
; rung 3
LD>=(325) D201 &9999  ; hours
UP(521)
MOV(021) &0 D201  ; hours

### Section Print

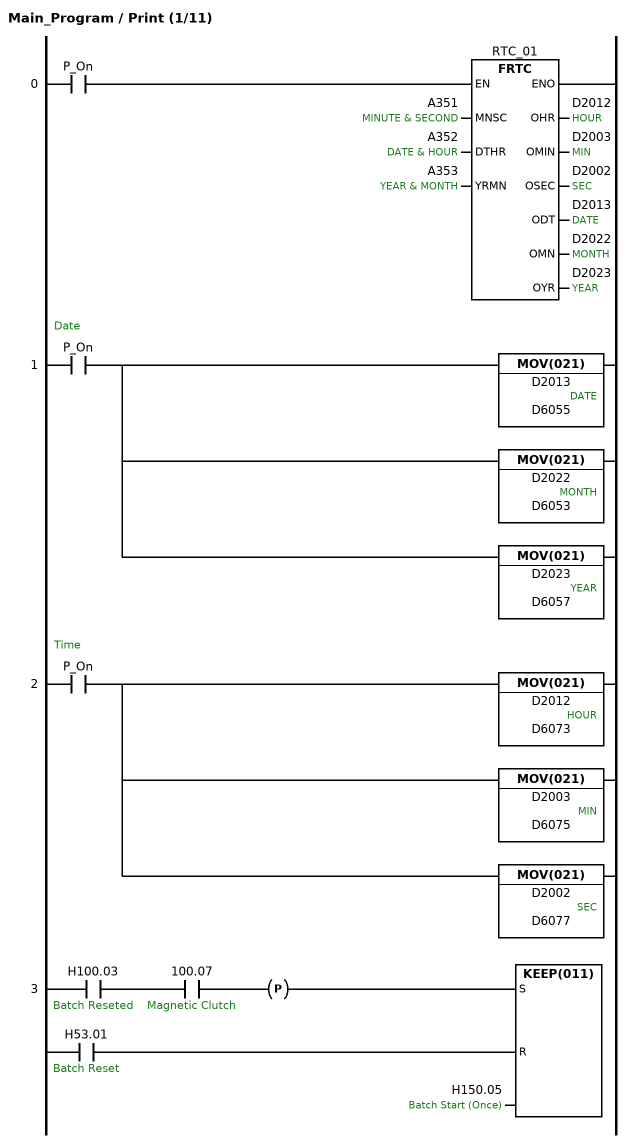
; rung 0
LD P_On
CALL RTC_01 : FRTC (MNSC := A351, DTHR := A352, YRMN := A353, OHR => D2012, OMIN => D2003, OSEC => D2002, ODT => D2013, OMN => D2022, OYR => D2023)  ; MINUTE & SECOND, DATE & HOUR, YEAR & MONTH, HOUR, MIN, SEC, DATE, MONTH, YEAR
; rung 1: Date
LD P_On
MOV(021) D2013 D6055  ; DATE
MOV(021) D2022 D6053  ; MONTH
MOV(021) D2023 D6057  ; YEAR
; rung 2: Time
LD P_On
MOV(021) D2012 D6073  ; HOUR
MOV(021) D2003 D6075  ; MIN
MOV(021) D2002 D6077  ; SEC
; rung 3
LD H100.03  ; Batch Reseted
AND 100.07  ; Magnetic Clutch
UP(521)
LD H53.01  ; Batch Reset
KEEP(011) H150.05  ; Batch Start (Once)

